(* CoDeSys 2.3.9.62 project: backupMain.pro *)
(* Libraries: BusDiag.lib, Standard.lib, Iecsfc.lib 8.11.10 11:37:48, SYSLIBCALLBACK.LIB *)

(* PLC configuration (modules and I/O channels)
K-Bus [K_Bus] node 0, in %IB0 out %QB0
input1 AT %IX0.0 [BOOLOnX_I] Ch_1 Digital input
input2 AT %IX0.1 [BOOLOnX_I] Ch_2 Digital input
input3 AT %IX0.2 [BOOLOnX_I] Ch_3 Digital input
input4 AT %IX0.3 [BOOLOnX_I] Ch_4 Digital input
input5 AT %IX0.4 [BOOLOnX_I] Ch_5 Digital input
input6 AT %IX0.5 [BOOLOnX_I] Ch_6 Digital input
input7 AT %IX0.6 [BOOLOnX_I] Ch_7 Digital input
input8 AT %IX0.7 [BOOLOnX_I] Ch_8 Digital input
outPut1 AT %QX0.0 [BOOLOnX_Q] Ch_1 Digital output
outPut2 AT %QX0.1 [BOOLOnX_Q] Ch_2 Digital output
AT %QX0.2 [BOOLOnX_Q] Ch_3 Digital output
AT %QX0.3 [BOOLOnX_Q] Ch_4 Digital output
AT %QX0.4 [BOOLOnX_Q] Ch_5 Digital output
AT %QX0.5 [BOOLOnX_Q] Ch_6 Digital output
AT %QX0.6 [BOOLOnX_Q] Ch_7 Digital output
AT %QX0.7 [BOOLOnX_Q] Ch_8 Digital output
Internal Digital I/O [InternalDigIO] node 1, in %IB512 out %QB512
  Internal Digital Inputs [Internal_DIN] node 0, in %IB512 out %QB512
    DIN1 AT %IX2300.0 [BOOLOnX_I] Internal Digital Input Bit 1
    DIN2 AT %IX2300.1 [BOOLOnX_I] Internal Digital Input Bit 2
  Internal Digital Outputs [Internal_DOUT] node 1, in %IB513 out %QB512
    DOUT1 AT %QX2300.0 [BOOLOnX_Q] Internal Digital Output Bit 1
    DOUT2 AT %QX2300.1 [BOOLOnX_Q] Internal Digital Output Bit 2
Fieldbus variables [FB_VARS] node 3, in %IB0 out %QB0
Flag variables [FLAG_VARS] node 4, in %IB0 out %QB0
Modbus-Master [MB_MASTER] node 5, in %IB0 out %QB0
*)

(* Task configuration *)
TASK main (PRIORITY := 15, INTERVAL := T#50ms);
	main();
END_TASK

(* POU main, ST *)
PROGRAM main
VAR
	roll : LREAL := 1;
	pitch : LREAL := 2;

	angle0 : LREAL;
	angle1 : LREAL;
	angle2 : LREAL;

	didBound : BOOL;

	angleFunction : ComputeMotorAngles;
	driverForMotor: MotorDriver;

	motorCounts: ARRAY[0..2] OF DINT;

	fromMotor: ARRAY[0..7] OF BYTE;

	toMotor0: BYTE;
	toMotor1: BYTE;
	toMotor2: BYTE;
	toMotor3: BYTE;
	toMotor4: BYTE;
	toMotor5: BYTE;
	toMotor6: BYTE;
	toMotor7: BYTE := 4;
	toMotor8: BYTE;

	DiagGetBusState : DiagGetBusState;
	gotData : BOOL;
END_VAR
fromMotor[0] := fromSlave0;
fromMotor[1] := fromSlave1;
fromMotor[2] := fromSlave2;
fromMotor[3] := fromSlave3;
fromMotor[4] := fromSlave4;
fromMotor[5] := fromSlave5;

toSlave0 := toMotor0;
toSlave1 := toMotor1;
toSlave2 := toMotor2;
toSlave3 := toMotor3;
toSlave4 := toMotor4;
toSlave5 := toMotor5;
toSlave6 := toMotor6;
toSlave7 := toMotor7;
toSlave8 := toMotor8;

DiagGetBusState.ENABLE := TRUE;
DiagGetBusState();


IF DiagGetBusState.READY THEN
	gotData := TRUE;
END_IF

angleFunction.roll := roll;
angleFunction.pitch := pitch;

angleFunction();

angle0 := angleFunction.angle0;
angle1 := angleFunction.angle1;
angle2 := angleFunction.angle2;
didBound := angleFunction.didBound;

driverForMotor.wantedMotor0 := angle0;
driverForMotor.wantedMotor1 := angle1;
driverForMotor.wantedMotor2 := angle2;
driverForMotor.endSwitchMotor0 := TRUE;
driverForMotor.endSwitchMotor1:= TRUE;
driverForMotor.endSwitchMotor2:= TRUE;

motorCounts[0] := driverForMotor.countsMotor0;
motorCounts[1] := driverForMotor.countsMotor1;
motorCounts[2] := driverForMotor.countsMotor2;
END_PROGRAM

(* POU ComputeMotorAngles, ST *)
FUNCTION_BLOCK ComputeMotorAngles
VAR_INPUT
	roll : LREAL;
	pitch : LREAL;
END_VAR
VAR_OUTPUT
	angle0 : LREAL;
	angle1 : LREAL;
	angle2 : LREAL;

	didBound : BOOL;
END_VAR
VAR
	l : LREAL := 1.75;
	delta : LREAL := 0.08;
	s0 : LREAL := 1.0;
	s1 : LREAL := 1.0;

	tmpVar : LREAL;

	p0 : LREAL;
	p1 : LREAL;
	p2 : LREAL;
END_VAR
tmpVar := l / 2 * ATAN(pitch / s1);
p1 :=delta + tmpVar;
p0 := delta - tmpVar;

p2 := delta - (l * SQRT(3) / 2) * ATAN(roll / s0);

p0 := -1.0 * (p0 - delta) / delta;
p1 := -1.0 * (p1 - delta) / delta;
p2 := -1.0 * (p2 - delta) / delta;

didBound := FALSE;

IF (p0 > 1.0) THEN
	p0 := 1.0;
	didBound := TRUE;
ELSIF (p0 < -1.0) THEN
	p0 := -1.0;
	didBound := TRUE;
END_IF


IF (p1 > 1.0) THEN
	p1 := 1.0;
	didBound := TRUE;
ELSIF (p1 < -1.0) THEN
	p1 := -1.0;
	didBound := TRUE;
END_IF

IF (p2 > 1.0) THEN
	p2 := 1.0;
	didBound := TRUE;
ELSIF (p2 < -1.0) THEN
	p2 := -1.0;
	didBound := TRUE;
END_IF

angle0 := ACOS(p0);
angle1 := ACOS(p1);
angle2 := ACOS(p2);
END_FUNCTION_BLOCK

(* POU MotorDriver, ST *)
FUNCTION_BLOCK MotorDriver
VAR_INPUT
	wantedMotor0: LREAL;
	wantedMotor1: LREAL;
	wantedMotor2: LREAL;
	endSwitchMotor0: BOOL;
	endSwitchMotor1: BOOL;
	endSwitchMotor2: BOOL;
END_VAR
VAR_OUTPUT
	countsMotor0: DINT;
	countsMotor1: DINT;
	countsMotor2: DINT;
END_VAR
VAR
	endSwitchPosition: DINT := -10000;
END_VAR
IF endSwitchMotor0 THEN
	countsMotor0 := motorAngleToCounts(wantedMotor0);
ELSE
	countsMotor0 := 0;
END_IF
IF endSwitchMotor0 THEN
	countsMotor1 := motorAngleToCounts(wantedMotor1);
ELSE
	countsMotor1 := 0;
END_IF
IF endSwitchMotor0 THEN
	countsMotor2 := motorAngleToCounts(wantedMotor2);
ELSE
	countsMotor2 := 0;
END_IF
END_FUNCTION_BLOCK

(* POU motorAngleToCounts, ST *)
FUNCTION motorAngleToCounts : DINT
VAR_INPUT
	wantedMotorAngle: LREAL;
END_VAR
VAR
	motorCountsPerRound: LREAL := 160000;
	pi: LREAL := 3.1415926;
	tempVar: INT;
END_VAR
motorAngleToCounts := REAL_TO_INT(LREAL_TO_REAL(wantedMotorAngle * motorCountsPerRound)/(2*pi)) - 10000;
END_FUNCTION

(* POU Configuration/MODBUS_CONFIGURATION, ST *)
PROGRAM MODBUS_CONFIGURATION        
VAR                                
END_VAR                            
(*
   <?xml version="1.0" encoding="UTF-16" standalone="yes"?>
<network xml_structure_version="1" xml_feature_version="1">
	<generator_settings minRTUTaskCycleTimeMs="5" minEthaskCycleTimeMs="5" ethSlaveMultiplier="0.1" rtuInterfaceMultiplier="0.1" taskGeneration="true"/>
</network>
                              
*)                                 
;
END_PROGRAM

(* POU UDPDecoder, ST *)
FUNCTION_BLOCK UDPDecoder
VAR_INPUT
	initialData: STRING(528);
END_VAR
VAR_OUTPUT
	floatArray : ARRAY [0..66] OF REAL;
END_VAR
VAR
   	hexSeperated: ARRAY[0..66] OF STRING(8);
	reversedHexSeperated: ARRAY[0..66] OF STRING(8);
	hexAsInt: ARRAY[0..66] OF REAL		(*Må være real for at EXPT funksjonen skal funke*);
	numberToMakeBinary: DWORD;
	binaryHexAsInt: ARRAY[0..66] OF ARRAY[0..31] OF BOOL;
 	i: INT;
	j: INT;
	k: INT;
	iterationCounter: INT := 0;
	calculationInt: INT;
	sign: INT;
	exponent: REAL;
	mantissa: REAL;
	hexArray: ARRAY[0..15] OF STRING(1);

END_VAR
(*Konvertering av little endian hexadecimal til flyttall*)
(*Usexy kode, finn ut hvordan det kan deklareres i deklareringsområdet*)
IF iterationCounter = 0 THEN
	hexArray[0] := '0';
	hexArray[1] := '1';
	hexArray[2] := '2';
	hexArray[3] := '3';
	hexArray[4] := '4';
	hexArray[5] := '5';
	hexArray[6] := '6';
	hexArray[7] := '7';
	hexArray[8] := '8';
	hexArray[9] := '9';
	hexArray[10] := 'a';
	hexArray[11] := 'b';
	hexArray[12] := 'c';
	hexArray[13] := 'd';
	hexArray[14] := 'e';
	hexArray[15] := 'f';

	(*Deler den oprinnlige tekststrengen opp i de forskjellige verdiene*)
	FOR i := 0 TO 66 DO
	    hexSeperated[i] := MID(initialData, 8, (i * 8) + 1);
	END_FOR

	(*Snur strengene for å passe med little endian*)
	FOR i := 0 TO 66 DO
		FOR j := 0 TO 7 BY 2 DO
			reversedHexSeperated[i] := CONCAT( reversedHexSeperated[i],  MID(hexSeperated[i], 2, 8 - j - 1));
		END_FOR
	END_FOR

	(*Regner ut  desimalen som hører til hexadesimalen*)
	FOR i := 0 TO 66 DO
		hexAsInt[i] := 0;
		FOR j := 0 TO 7 DO
			FOR k := 0 TO 15 DO
				IF MID(reversedHexSeperated[i], 1, j + 1) = hexArray[k] THEN
					hexAsInt[i] := hexAsInt[i] + k * EXPT(16, 7 - j);
					EXIT;
				END_IF
			END_FOR
		END_FOR
	END_FOR

	(*Gjør inten om til binært for å kunne regne ut mantissa, eksponent og sign*)
	FOR i := 0 TO 66 DO
		numberToMakeBinary := REAL_TO_DWORD(hexAsInt[i]);
		FOR j := 0 TO 31 DO
			binaryHexAsInt[i][j] := (numberToMakeBinary AND 16#80000000) <> 0;
			numberToMakeBinary := SHL(numberToMakeBinary, 1);
		END_FOR
	END_FOR

	(*Regner ut sign, eksponent og mantissa*)
	FOR i := 0 TO 66 DO
		sign := 0;
		exponent := 0;
		mantissa := 0;
		(*Sjekker første binærtallet for å finne ut om det er positivt eller negativt*)
		IF NOT binaryHexAsInt[i][0] THEN
			sign := 0;
		ELSE
			sign := 1;
		END_IF
		(*Regner ut eksponenten for fra binærtallet*)
		FOR j := 1 TO 8 DO
            		IF binaryHexAsInt[i][j] THEN
                		exponent := exponent + EXPT(2, 8 - j);
	            END_IF
        	END_FOR
        	exponent := exponent - 127;
		(*Regner ut mantissaen med de resterende talla i binærtallet*)
		FOR j := 9 TO 31 DO
            		IF binaryHexAsInt[i][j] THEN
                		mantissa := mantissa + EXPT(2, 8 - j);
	            END_IF
       	 END_FOR

		floatArray[i] := EXPT(-1, sign) * (1.0 + mantissa) * EXPT(2, exponent);
	END_FOR

	iterationCounter := iterationCounter + 1;
END_IF
END_FUNCTION_BLOCK
